TYPE MotorInputVariables :
STRUCT
	Start : BOOL;
	Stop : BOOL;
	Oveload : BOOL;
END_STRUCT
END_TYPE

(* stored: Version 1.1.0.1, ProductVersion 3.1.4024.9
   DUT MotorInputVariables: Id {aa82066d-e38e-4fac-b31b-9058e8869ac4} *)
